(* IEC 61131-3 sources: AutomationLab/ConveyorObject/Model, 2 files *)

(* ---- Conveyer1.st ---- *)
FUNCTION_BLOCK Conveyer1
VAR
    // Логический блок управления лентой конвейера
    logic: LogicDevice;
END_VAR
VAR_IN_OUT
    // Данные технологического объекта конвейера
    Data: ConveyorType;
END_VAR

// ============================================
// УСТРОЙСТВО — МОДЕЛЬ УПРАВЛЕНИЯ КОНВЕЙЕРОМ
// ============================================
// Принимает данные с датчиков через структуру ConveyorType,
// вызывает логику принятия решения (LogicDevice)
// и записывает команду на вращение ленты обратно в структуру.
// ============================================

// Логика: появление коробки на старте запускает ленту,
// достижение конца — останавливает
logic(BoxOnStart:= Data.BoxOnStartPosition, BoxOnEnd:= Data.BoxOnEndPosition, ComRotate=> Data.ComRotateBelt);

(* ---- Conveyor.st ---- *)
FUNCTION_BLOCK Conveyor
VAR_INPUT
END_VAR
VAR_OUTPUT
END_VAR
VAR
END_VAR
VAR_IN_OUT
	Data: ConveyorType;
END_VAR

Data.ComRotateBelt := AlwaysOn(Allow := NOT Data.BoxOnEndPosition);
